(* IEC 61131-3 sources: brdkAGV_PLC/vsCode/ros_topics_typ/ros_topics, 1 file *)

(* ---- ros_topics.fun ---- *)
FUNCTION_BLOCK ros_topics_typInit
	VAR_OUTPUT
		Handle : UDINT;
	END_VAR
	VAR
		_state : USINT;
	END_VAR
END_FUNCTION_BLOCK

FUNCTION_BLOCK ros_topics_typCyclic
	VAR_INPUT
		Enable : BOOL;
		Handle : UDINT;
		Start : BOOL;
		pros_topics_typ : REFERENCE TO ros_topics_typ;
	END_VAR
	VAR_OUTPUT
		Active : BOOL;
		Error : BOOL;
		Disconnected : BOOL;
		Connected : BOOL;
		Operational : BOOL;
		Aborted : BOOL;
	END_VAR
	VAR
		_state : USINT;
	END_VAR
END_FUNCTION_BLOCK

FUNCTION_BLOCK ros_topics_typExit
	VAR_INPUT
		Handle : UDINT;
	END_VAR
	VAR
		_state : USINT;
	END_VAR
END_FUNCTION_BLOCK
